// TIA Portal V17 export
// export: Created 2025-03-05T08:03:43.2074788Z, ExportSetting WithDefaults, DisplayName Totally Integrated Automation Portal, DisplayVersion V17 Update 8, DisplayName TIA Portal Openness, DisplayVersion V17 Update 8, DisplayName TIA Portal Version Control Interface, DisplayVersion V17, DisplayName SINAMICS Startdrive Advanced, DisplayVersion V17 SP2, DisplayName SINAMICS Startdrive G110M, G120, G120C, G120D, G120P, G115D, DisplayVersion V17 SP2, DisplayName SINAMICS Startdrive G130, G150, S120, S150, SINAMICS MV, S210, DisplayVersion V17 SP2, DisplayName STEP 7 Professional, DisplayVersion V17 Update 8, DisplayName SINUMERIK ONE STEP 7 Toolbox, DisplayVersion V17 Update 12, DisplayName SINUMERIK 840D sl STEP 7 Toolbox, DisplayVersion V17 Update 12, DisplayName STEP 7 Safety, DisplayVersion V17 Update 6, DisplayName WinCC Advanced, DisplayVersion V17 Update 8
TYPE "HMI_DATA_START_STOP"
// stored: IsFailsafeCompliant false
   STRUCT
      HMI_START : Bool;   // HMI start
      HMI_STOP : Bool;   // HMI stop
      HMI_STARTED : Bool;   // HMI started
      HMI_STOPPED : Bool;   // HMI stopped
      HMI_STARTING : Bool;   // HMI starting
      HMI_STOPPING : Bool;   // HMI stopping
      HMI_START_CONDITIONS : Bool;   // HMI start conditions
      HMI_STOP_CONDITIONS : Bool;   // HMI stop conditions
   END_STRUCT;
END_TYPE
